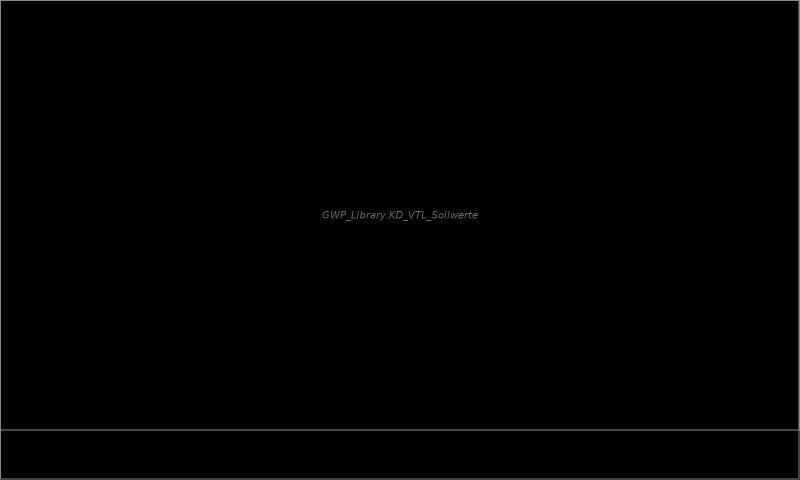
VISUALIZATION KD_VTL_Sollwerte  // 800x480
    Frame (0,0 800x430)
        shows GWP_Library.KD_VTL_Sollwerte(FB_KD := Main.KD_0, FB_Init_1 := Main.Init_0)
END_VISUALIZATION

(* stored: Version 1.1.0.1, ProductVersion 3.1.4022.6
   Visu KD_VTL_Sollwerte: Id {b1ab3118-89e0-43a0-8067-5c8ba679c9af} *)
